// TIA Portal V17 export
// export: Created 2022-05-07T16:38:48.4672323Z, ExportSetting WithDefaults, DisplayName Totally Integrated Automation Portal, DisplayVersion V17 Update 3, DisplayName TIA Portal Openness, DisplayVersion V17 Update 3, DisplayName TIA Portal Version Control Interface, DisplayVersion V17, DisplayName TIA Portal Test Suite Advanced, DisplayVersion V17 Update 1, DisplayName SINAMICS Startdrive Advanced, DisplayVersion V17 Update2, DisplayName SINAMICS Startdrive G130, G150, S120, S150, SINAMICS MV, S210, DisplayVersion V17 Update2, DisplayName SINAMICS Startdrive G110M, G120, G120C, G120D, G120P, G115D, DisplayVersion V17 Update2, DisplayName STEP 7 Professional, DisplayVersion V17 Update 3, DisplayName STEP 7 Safety, DisplayVersion V17, DisplayName WinCC UA Professional, DisplayVersion V17 Update 3
DATA_BLOCK "DBParAssi"   // DB12
{ S7_Optimized_Access := 'TRUE' }
VERSION : 0.1
// stored: AutoNumber true, DBAccessibleFromOPCUA true, IsOnlyStoredInLoadMemory false, IsRetainMemResEnabled false, IsWriteProtectedInAS false, MemoryReserve 100
   VAR RETAIN
      MR : "UDTMotori";
      MA { S7_SetPoint := 'True'} : "UDTMotori";
      MS { S7_SetPoint := 'True'} : "UDTMotori";
      ME { S7_SetPoint := 'True'} : "UDTMotori";
   END_VAR
BEGIN
   MR.pos."1" := 120.0;   // [°] predisposizione (detorsione)
   MR.pos."2" := 10.0;   // [°] quota intermedia (detorsione parziale) / [°] quota intermedia
   MR.pos."3" := 0.0;   // [°] zero / [°]
   MR.pos."4" := 180.0;   // [°] ritorsione
   MR.vel."1" := 1000.0;   // [°/s] vel detorsione
   MR.vel."2" := 1000.0;   // [°/s] vel detorsione parziale
   MR.vel."3" := 200.0;   // [°/s] vel
   MR.vel."4" := 200.0;   // [°/s] vel ritorsione
   MR.IN.Sp_Jog_Velocity := 80.0;
   MR.IN.Sp_MoveRel_Velocity := 1000.0;
   MR.IN.Sp_MoveAbs_Velocity := 1000.0;
   MR.IN.Sp_RampUpTime := 2.0;
   MR.IN.Sp_RampDnTime := 2.0;
   MA.pos."1" := 7.5;   // [mm] quota detorsione / [mm]
   MA.pos."2" := 12.5;   // [mm] quota fissa era 12.5 / [mm]
   MA.pos."3" := 9.6;   // [mm] quota ritorsione / [mm]
   MA.pos."4" := 0.0;   // [mm]
   MA.IN.Sp_Jog_Velocity := 5.0;
   MA.IN.Sp_MoveRel_Velocity := 150.0;
   MA.IN.Sp_MoveAbs_Velocity := 50.0;
   MS.pos."1" := 220.0;   // [pulses] preset (800 0 giro completo) / [pulses] preset (400 0 giro completo)
   // MS.pos."2" : [pulses]
   MS.pos."3" := 95.0;   // [p] quota MA
   MS.vel."1" := 3000.0;   // [p/s]
   MS.vel."3" := 3000.0;   // [p/s]
   MS.IN.Sp_Jog_Velocity := 180.0;
   MS.IN.Sp_MoveRel_Distance := 230.0;
   MS.IN.Sp_MoveRel_Velocity := 1000.0;
   MS.IN.Sp_MoveAbs_Velocity := 1000.0;
   ME.pos."1" := 120.0;   // [°] quota blocco fili / [°]
   ME.pos."2" := 0.0;   // [°] Home position / [°]
   ME.IN.Sp_Jog_Velocity := 200.0;
   ME.IN.Sp_MoveRel_Velocity := 1000.0;
   ME.IN.Sp_MoveAbs_Velocity := 1000.0;
END_DATA_BLOCK
